TYPE ST_EAPMachineState : 
	STRUCT
		(* Comando in esecuzione *)
		Cmd : UDINT;
		(* Stato del comando in esecuzione *)
		CmdCase : UDINT;
		(* Errore generico della Macchina *)
		Error : UDINT;
		(* Errore specifico della Macchina *)
		ErrorExtra : UDINT;
		(* Macchina con potenza attiva *)
		PowerActive : BOOL;
		(* Macchina con Home eseguito *)
		Homed : BOOL;
		(* Macchina in automatico *)
		Auto : BOOL;
		(* Macchina in automatico e con ciclo di lavoro attivo -> sta lavorando *)
		Working : BOOL;
		(* Macchina accesso manuale in area segreta attivo *)
		ManAccesActive : BOOL;
		(* Macchina in Emergenza *)
		EmergencyOK : BOOL;
	END_STRUCT
END_TYPE

(* stored: Version 1.1.0.1, ProductVersion 3.1.4024.11
   DUT ST_EAPMachineState: Id {2c4c196f-0f6c-4fc5-8656-d0e5b1b8a202} *)
